Omron Sysmac Studio project Compare_Examp (Sysmac Studio 1.65.0.64007, StandardProject)

# Controller new_Controller_0: NX1P2-1040DT1 version 1.69
Task PrimaryTask (priority 4, period or condition 2000): Program0

VAR_GLOBAL
    BIO_Input_Bit_00 : BOOL;  (* at BuiltInIO://cpu/#0/Input_Bit_00 *)
    BIO_Input_Bit_01 : BOOL;  (* at BuiltInIO://cpu/#0/Input_Bit_01 *)
    BIO_Output_Bit_00 : BOOL;  (* at BuiltInIO://cpu/#0/Output_Bit_00 *)
    BIO_Output_Bit_01 : BOOL;  (* at BuiltInIO://cpu/#0/Output_Bit_01 *)
    BIO_Output_Bit_02 : BOOL;  (* at BuiltInIO://cpu/#0/Output_Bit_02 *)
    Start : BOOL;
    Stop : BOOL;
    OUT_MikserMotor_Start : BOOL;
    OUT_P1_Valf : BOOL;
    OUT_P2_Valf : BOOL;
    OUT_P3_Valf : BOOL;
    IN_Start_Button : BOOL;
    IN_Stop_Button : BOOL;
    Sistem_Calisiyor : BOOL;
    SistemCalismaSuresi|Reset : BOOL;
    SistemCalismaSuresi_Reset : BOOL;
END_VAR

PROGRAM Program0
VAR
    SistemCalismaSuresi : AccumulationTimer;
    SistemCalismaSuresi_ET : TIME;
END_VAR
VAR_EXTERNAL
    BIO_Input_Bit_00 : BOOL;
    BIO_Input_Bit_01 : BOOL;
    Start : BOOL;
    Stop : BOOL;
    OUT_MikserMotor_Start : BOOL;
    BIO_Output_Bit_00 : BOOL;
    OUT_P1_Valf : BOOL;
    BIO_Output_Bit_01 : BOOL;
    OUT_P2_Valf : BOOL;
    OUT_P3_Valf : BOOL;
    BIO_Output_Bit_02 : BOOL;
    IN_Start_Button : BOOL;
    IN_Stop_Button : BOOL;
    Sistem_Calisiyor : BOOL;
    SistemCalismaSuresi|Reset : BOOL;
    SistemCalismaSuresi_Reset : BOOL;
END_VAR
VAR
    _p1 : BOOL;
END_VAR

(* Section Section0: ladder, written here as Structured Text *)

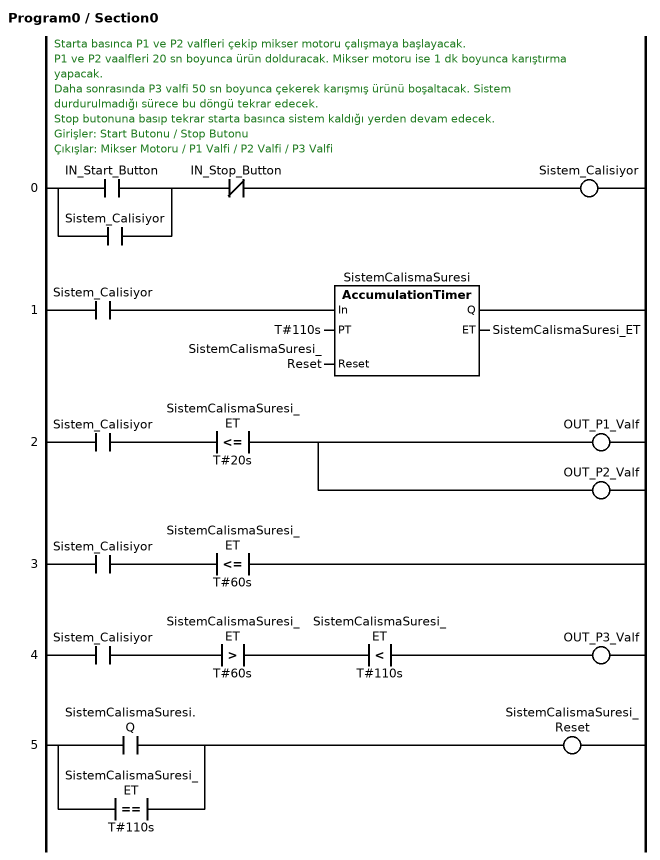
(* Rung 0: Starta basınca P1 ve P2 valfleri çekip mikser motoru çalışmaya başlayacak. / P1 ve P2 vaalfleri 20 sn boyunca ürün dolduracak. Mikser motoru ise 1 dk boyunca karıştırma yapacak. / Daha sonrasında P3 valfi 50 sn boyunca çekerek karışmış ürünü boşaltacak. Sistem durdurulmadığı sürece bu döngü tekrar edecek. / Stop butonuna basıp tekrar starta basınca sistem kaldığı yerden devam edecek. / Girişler: Start Butonu / Stop Butonu / Çıkışlar: Mikser Motoru / P1 Valfi / P2 Valfi / P3 Valfi *)
Sistem_Calisiyor := (IN_Start_Button OR Sistem_Calisiyor) AND NOT IN_Stop_Button;
(* Rung 1 *)
SistemCalismaSuresi(In := Sistem_Calisiyor, PT := T#110s, Reset := SistemCalismaSuresi_Reset, ET => SistemCalismaSuresi_ET);
(* Rung 2 *)
_p1 := Sistem_Calisiyor AND (SistemCalismaSuresi_ET <= T#20s);
OUT_P1_Valf := _p1;
OUT_P2_Valf := _p1;
(* Rung 3 *)
(* drawn but driving nothing: Sistem_Calisiyor, SistemCalismaSuresi_ET, T#60s *)
(* Rung 4 *)
OUT_P3_Valf := Sistem_Calisiyor AND (SistemCalismaSuresi_ET > T#60s) AND (SistemCalismaSuresi_ET < T#110s);
(* Rung 5 *)
SistemCalismaSuresi_Reset := SistemCalismaSuresi.Q OR (SistemCalismaSuresi_ET = T#110s);

(* Section InOut: ladder, written here as Structured Text *)

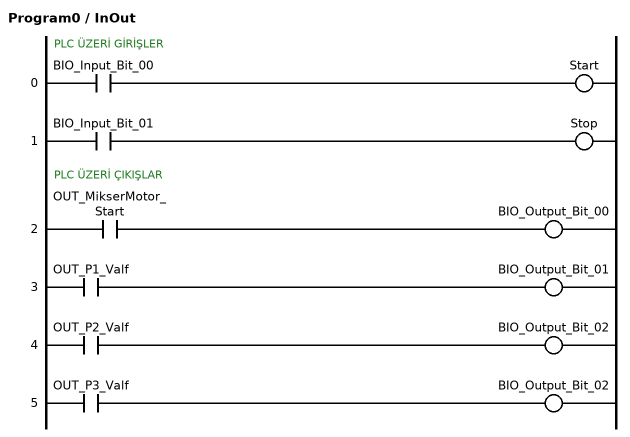
(* Rung 0: PLC ÜZERİ GİRİŞLER *)
Start := BIO_Input_Bit_00;
(* Rung 1 *)
Stop := BIO_Input_Bit_01;
(* Rung 2: PLC ÜZERİ ÇIKIŞLAR *)
BIO_Output_Bit_00 := OUT_MikserMotor_Start;
(* Rung 3 *)
BIO_Output_Bit_01 := OUT_P1_Valf;
(* Rung 4 *)
BIO_Output_Bit_02 := OUT_P2_Valf;
(* Rung 5 *)
BIO_Output_Bit_02 := OUT_P3_Valf;
END_PROGRAM